FUNCTION_BLOCK FB_PTOStepperRotate
VAR_INPUT
	bExecute	: BOOL;
	bStop		: BOOL;
	bCCW		: BOOL;	//Gegen Uhrzeiger
	nSpeed		: UINT;	//Steps/sec
END_VAR
VAR_OUTPUT
	bBusy		: BOOL;
END_VAR
VAR_IN_OUT
	pPTOStepperRef : POINTER TO ST_PTOStepperRef;
END_VAR
VAR
	nSpeedIntern : INT;
	nState : USINT;
END_VAR

IF bExecute THEN
	CASE nState OF
		0:	//Prepare
			IF bStop THEN
				RETURN;
			END_IF
			bBusy := TRUE;
			IF bCCW THEN
				nSpeedIntern := UINT_TO_INT(nSpeed);
			ELSE
				nSpeedIntern := -UINT_TO_INT(nSpeed);
			END_IF
			MEMCPY(ADR(pPTOStepperRef^.nFrequencyValue),ADR(nSpeedIntern),2);
			nState := 1;
			
		1:	//Waiting for stop
			IF bStop THEN
				pPTOStepperRef^.nFrequencyValue := 0;
				nState := 80;
				bBusy := FALSE;
			END_IF
	END_CASE
ELSE
	nState := 0;
	bBusy := FALSE;	
END_IF

END_FUNCTION_BLOCK

(* stored: Version 1.1.0.1, ProductVersion 3.1.4020.12
   POU FB_PTOStepperRotate: Id {d78bdff1-196a-40e4-bc79-b7c42aa8dd96}, SpecialFunc None *)
